# EPICS substitutions: db/MLoutput.substitutions
file "/epics/iocs/MachineLearn/db/MLoutput_sub.db"
{
pattern
{CELL, WIRE}
{"01", "33"}
{"01", "34"}
{"01", "35"}
{"01", "36"}
{"01", "37"}
{"01", "38"}
{"01", "39"}
{"01", "40"}
{"01", "41"}
{"01", "42"}
{"01", "43"}
{"01", "44"}
{"01", "45"}
{"01", "46"}
{"01", "47"}
{"01", "48"}
{"01", "49"}
{"01", "50"}
{"01", "51"}
{"01", "52"}

{"02", "33"}
{"02", "34"}
{"02", "35"}
{"02", "36"}
{"02", "37"}
{"02", "38"}
{"02", "39"}
{"02", "40"}
{"02", "41"}
{"02", "42"}
{"02", "43"}
{"02", "44"}
{"02", "45"}
{"02", "46"}
{"02", "47"}
{"02", "48"}
{"02", "49"}
{"02", "50"}
{"02", "51"}
{"02", "52"}

{"03", "55"}
{"03", "56"}
{"03", "57"}
{"03", "58"}
{"03", "59"}
{"03", "60"}
{"03", "61"}
{"03", "62"}
{"03", "63"}
{"03", "64"}
{"03", "65"}
{"03", "66"}
{"03", "67"}
{"03", "68"}
{"03", "69"}
{"03", "70"}
{"03", "71"}
{"03", "72"}
{"03", "73"}
{"03", "74"}

{"04", "33"}
{"04", "34"}
{"04", "35"}
{"04", "36"}
{"04", "37"}
{"04", "38"}
{"04", "39"}
{"04", "40"}
{"04", "41"}
{"04", "42"}
{"04", "43"}
{"04", "44"}
{"04", "45"}
{"04", "46"}
{"04", "47"}
{"04", "48"}
{"04", "49"}
{"04", "50"}
{"04", "51"}
{"04", "52"}

{"05", "33"}
{"05", "34"}
{"05", "35"}
{"05", "36"}
{"05", "37"}
{"05", "38"}
{"05", "39"}
{"05", "40"}
{"05", "41"}
{"05", "42"}
{"05", "43"}
{"05", "44"}
{"05", "45"}
{"05", "46"}
{"05", "47"}
{"05", "48"}
{"05", "49"}
{"05", "50"}
{"05", "51"}
{"05", "52"}

{"06", "33"}
{"06", "34"}
{"06", "35"}
{"06", "36"}
{"06", "37"}
{"06", "38"}
{"06", "39"}
{"06", "40"}
{"06", "41"}
{"06", "42"}
{"06", "43"}
{"06", "44"}
{"06", "45"}
{"06", "46"}
{"06", "47"}
{"06", "48"}
{"06", "49"}
{"06", "50"}
{"06", "51"}
{"06", "52"}

{"07", "33"}
{"07", "34"}
{"07", "35"}
{"07", "36"}
{"07", "37"}
{"07", "38"}
{"07", "39"}
{"07", "40"}
{"07", "41"}
{"07", "42"}
{"07", "43"}
{"07", "44"}
{"07", "45"}
{"07", "46"}
{"07", "47"}
{"07", "48"}
{"07", "49"}
{"07", "50"}
{"07", "51"}
{"07", "52"}

{"08", "33"}
{"08", "34"}
{"08", "35"}
{"08", "36"}
{"08", "37"}
{"08", "38"}
{"08", "39"}
{"08", "40"}
{"08", "41"}
{"08", "42"}
{"08", "43"}
{"08", "44"}
{"08", "45"}
{"08", "46"}
{"08", "47"}
{"08", "48"}
{"08", "49"}
{"08", "50"}
{"08", "51"}
{"08", "52"}

{"09", "33"}
{"09", "34"}
{"09", "35"}
{"09", "36"}
{"09", "37"}
{"09", "38"}
{"09", "39"}
{"09", "40"}
{"09", "41"}
{"09", "42"}
{"09", "43"}
{"09", "44"}
{"09", "45"}
{"09", "46"}
{"09", "47"}
{"09", "48"}
{"09", "49"}
{"09", "50"}
{"09", "51"}
{"09", "52"}

{"10", "33"}
{"10", "34"}
{"10", "35"}
{"10", "36"}
{"10", "37"}
{"10", "38"}
{"10", "39"}
{"10", "40"}
{"10", "41"}
{"10", "42"}
{"10", "43"}
{"10", "44"}
{"10", "45"}
{"10", "46"}
{"10", "47"}
{"10", "48"}
{"10", "49"}
{"10", "50"}
{"10", "51"}
{"10", "52"}

{"11", "33"}
{"11", "34"}
{"11", "35"}
{"11", "36"}
{"11", "37"}
{"11", "38"}
{"11", "39"}
{"11", "40"}
{"11", "41"}
{"11", "42"}
{"11", "43"}
{"11", "44"}
{"11", "45"}
{"11", "46"}
{"11", "47"}
{"11", "48"}
{"11", "49"}
{"11", "50"}
{"11", "51"}
{"11", "52"}

{"12", "33"}
{"12", "34"}
{"12", "35"}
{"12", "36"}
{"12", "37"}
{"12", "38"}
{"12", "39"}
{"12", "40"}
{"12", "41"}
{"12", "42"}
{"12", "43"}
{"12", "44"}
{"12", "45"}
{"12", "46"}
{"12", "47"}
{"12", "48"}
{"12", "49"}
{"12", "50"}
{"12", "51"}
{"12", "52"}

{"13", "33"}
{"13", "34"}
{"13", "35"}
{"13", "36"}
{"13", "37"}
{"13", "38"}
{"13", "39"}
{"13", "40"}
{"13", "41"}
{"13", "42"}
{"13", "43"}
{"13", "44"}
{"13", "45"}
{"13", "46"}
{"13", "47"}
{"13", "48"}
{"13", "49"}
{"13", "50"}
{"13", "51"}
{"13", "52"}
{"13", "53"}
{"13", "54"}
{"13", "55"}
{"13", "56"}

{"14", "33"}
{"14", "34"}
{"14", "35"}
{"14", "36"}
{"14", "37"}
{"14", "38"}
{"14", "39"}
{"14", "40"}
{"14", "41"}
{"14", "42"}
{"14", "43"}
{"14", "44"}
{"14", "45"}
{"14", "46"}
{"14", "47"}
{"14", "48"}
{"14", "49"}
{"14", "50"}
{"14", "51"}
{"14", "52"}

{"15", "33"}
{"15", "34"}
{"15", "35"}
{"15", "36"}
{"15", "37"}
{"15", "38"}
{"15", "39"}
{"15", "40"}
{"15", "41"}
{"15", "42"}
{"15", "43"}
{"15", "44"}
{"15", "45"}
{"15", "46"}
{"15", "47"}
{"15", "48"}
{"15", "49"}
{"15", "50"}
{"15", "51"}
{"15", "52"}

{"16", "33"}
{"16", "34"}
{"16", "35"}
{"16", "36"}
{"16", "37"}
{"16", "38"}
{"16", "39"}
{"16", "40"}
{"16", "41"}
{"16", "42"}
{"16", "43"}
{"16", "44"}
{"16", "45"}
{"16", "46"}
{"16", "47"}
{"16", "48"}
{"16", "49"}
{"16", "50"}
{"16", "51"}
{"16", "52"}

{"17", "36"}
{"17", "37"}
{"17", "38"}
{"17", "39"}
{"17", "40"}
{"17", "41"}
{"17", "42"}
{"17", "43"}
{"17", "44"}
{"17", "45"}
{"17", "46"}
{"17", "47"}
{"17", "48"}
{"17", "49"}
{"17", "50"}
{"17", "51"}
{"17", "52"}
{"17", "53"}
{"17", "54"}
{"17", "55"}
{"17", "56"}
{"17", "57"}
{"17", "58"}
{"17", "59"}

{"18", "33"}
{"18", "34"}
{"18", "35"}
{"18", "36"}
{"18", "37"}
{"18", "38"}
{"18", "39"}
{"18", "40"}
{"18", "41"}
{"18", "42"}
{"18", "43"}
{"18", "44"}
{"18", "45"}
{"18", "46"}
{"18", "47"}
{"18", "48"}
{"18", "49"}
{"18", "50"}
{"18", "51"}
{"18", "52"}
{"18", "53"}
{"18", "54"}
{"18", "55"}
{"18", "56"}

{"19", "33"}
{"19", "34"}
{"19", "35"}
{"19", "36"}
{"19", "37"}
{"19", "38"}
{"19", "39"}
{"19", "40"}
{"19", "41"}
{"19", "42"}
{"19", "43"}
{"19", "44"}
{"19", "45"}
{"19", "46"}
{"19", "47"}
{"19", "48"}
{"19", "49"}
{"19", "50"}
{"19", "51"}
{"19", "52"}
{"19", "53"}
{"19", "54"}
{"19", "55"}
{"19", "56"}

{"20", "33"}
{"20", "34"}
{"20", "35"}
{"20", "36"}
{"20", "37"}
{"20", "38"}
{"20", "39"}
{"20", "40"}
{"20", "41"}
{"20", "42"}
{"20", "43"}
{"20", "44"}
{"20", "45"}
{"20", "46"}
{"20", "47"}
{"20", "48"}
{"20", "49"}
{"20", "50"}
{"20", "51"}
{"20", "52"}

{"21", "33"}
{"21", "34"}
{"21", "35"}
{"21", "36"}
{"21", "37"}
{"21", "38"}
{"21", "39"}
{"21", "40"}
{"21", "41"}
{"21", "42"}
{"21", "43"}
{"21", "44"}
{"21", "45"}
{"21", "46"}
{"21", "47"}
{"21", "48"}
{"21", "49"}
{"21", "50"}
{"21", "51"}
{"21", "52"}

{"22", "33"}
{"22", "34"}
{"22", "35"}
{"22", "36"}
{"22", "37"}
{"22", "38"}
{"22", "39"}
{"22", "40"}
{"22", "41"}
{"22", "42"}
{"22", "43"}
{"22", "44"}
{"22", "45"}
{"22", "46"}
{"22", "47"}
{"22", "48"}
{"22", "49"}
{"22", "50"}
{"22", "51"}
{"22", "52"}

{"23", "33"}
{"23", "34"}
{"23", "35"}
{"23", "36"}
{"23", "37"}
{"23", "38"}
{"23", "39"}
{"23", "40"}
{"23", "41"}
{"23", "42"}
{"23", "43"}
{"23", "44"}
{"23", "45"}
{"23", "46"}
{"23", "47"}
{"23", "48"}
{"23", "49"}
{"23", "50"}
{"23", "51"}
{"23", "52"}
{"23", "53"}
{"23", "54"}
{"23", "55"}
{"23", "56"}

{"24", "33"}
{"24", "34"}
{"24", "35"}
{"24", "36"}
{"24", "37"}
{"24", "38"}
{"24", "39"}
{"24", "40"}
{"24", "41"}
{"24", "42"}
{"24", "43"}
{"24", "44"}
{"24", "45"}
{"24", "46"}
{"24", "47"}
{"24", "48"}
{"24", "49"}
{"24", "50"}
{"24", "51"}
{"24", "52"}

{"25", "33"}
{"25", "34"}
{"25", "35"}
{"25", "36"}
{"25", "37"}
{"25", "38"}
{"25", "39"}
{"25", "40"}
{"25", "41"}
{"25", "42"}
{"25", "43"}
{"25", "44"}
{"25", "45"}
{"25", "46"}
{"25", "47"}
{"25", "48"}
{"25", "49"}
{"25", "50"}
{"25", "51"}
{"25", "52"}

{"26", "33"}
{"26", "34"}
{"26", "35"}
{"26", "36"}
{"26", "37"}
{"26", "38"}
{"26", "39"}
{"26", "40"}
{"26", "41"}
{"26", "42"}
{"26", "43"}
{"26", "44"}
{"26", "45"}
{"26", "46"}
{"26", "47"}
{"26", "48"}
{"26", "49"}
{"26", "50"}
{"26", "51"}
{"26", "52"}

{"27", "33"}
{"27", "34"}
{"27", "35"}
{"27", "36"}
{"27", "37"}
{"27", "38"}
{"27", "39"}
{"27", "40"}
{"27", "41"}
{"27", "42"}
{"27", "43"}
{"27", "44"}
{"27", "45"}
{"27", "46"}
{"27", "47"}
{"27", "48"}
{"27", "49"}
{"27", "50"}
{"27", "51"}
{"27", "52"}

{"28", "33"}
{"28", "34"}
{"28", "35"}
{"28", "36"}
{"28", "37"}
{"28", "38"}
{"28", "39"}
{"28", "40"}
{"28", "41"}
{"28", "42"}
{"28", "43"}
{"28", "44"}
{"28", "45"}
{"28", "46"}
{"28", "47"}
{"28", "48"}
{"28", "49"}
{"28", "50"}
{"28", "51"}
{"28", "52"}

{"29", "33"}
{"29", "34"}
{"29", "35"}
{"29", "36"}
{"29", "37"}
{"29", "38"}
{"29", "39"}
{"29", "40"}
{"29", "41"}
{"29", "42"}
{"29", "43"}
{"29", "44"}
{"29", "45"}
{"29", "46"}
{"29", "47"}
{"29", "48"}
{"29", "49"}
{"29", "50"}
{"29", "51"}
{"29", "52"}

{"30", "33"}
{"30", "34"}
{"30", "35"}
{"30", "36"}
{"30", "37"}
{"30", "38"}
{"30", "39"}
{"30", "40"}
{"30", "41"}
{"30", "42"}
{"30", "43"}
{"30", "44"}
{"30", "45"}
{"30", "46"}
{"30", "47"}
{"30", "48"}
{"30", "49"}
{"30", "50"}
{"30", "51"}
{"30", "52"}
}
